FUNCTION_BLOCK FB_RepetitionRate
VAR_INPUT
	frequencyRaw : UDINT;
END_VAR
VAR_OUTPUT
	Inhibit : BOOL;
	AboveThreshold : BOOL;
END_VAR
VAR
	RepetitionRateHz : REAL;
END_VAR
VAR CONSTANT
	ScalingFactor: REAL := 100; // Scaling of raw input frequency
	Threshold : REAL := 10.0; // set this for determening AboveThreshold
END_VAR


//check the card how to scale the input and how to set the frequency in configuration
RepetitionRateHz := UDINT_TO_REAL(frequencyRaw)/ScalingFactor;

AboveThreshold := RepetitionRateHz > Threshold;

METHOD Control : BOOL
VAR_IN_OUT
	structure : ST_RepetitionRate;
END_VAR
structure.RepetitionRateHzSt := RepetitionRateHz;
structure.RepRateAboveThresholdSt := AboveThreshold;
structure.RepetitionRateHzThreshold := Threshold;
END_METHOD

END_FUNCTION_BLOCK

(* stored: Version 1.1.0.1, ProductVersion 3.1.4024.12
   POU FB_RepetitionRate: Id {423750c0-d8f4-43bf-b0d4-b19db13c840f}, SpecialFunc None
   Method Control: Id {2f00e7fb-7844-4f70-857f-b164c8112c6a} *)
